(* CODESYS project AULA1.project

Project tree, tasks and I/O mapping:
  Device : CODESYS Control Win V3, 3S - Smart Software Solutions GmbH, order no. 305021, version 3.5.11.30
    application Application
      libraries: Standard, * (System)
      task MainTask (cyclic, interval t#20ms, priority 1) calls PLC_PRG
      task VISU_TASK (cyclic, interval 100 ms, priority 31) calls VisuElems.Visu_Prg
      program PLC_PRG [LD]
      visualisation Visualization
  text list GlobalTextList
*)

// Device/Application/PLC_PRG
PROGRAM PLC_PRG
VAR
	A : BOOL;
	B : BOOL;
	C : BOOL;
	SNOT: BOOL;
	SOR: BOOL;
	SAND2: BOOL;
	SAND1: BOOL;
	SA : BOOL;
END_VAR

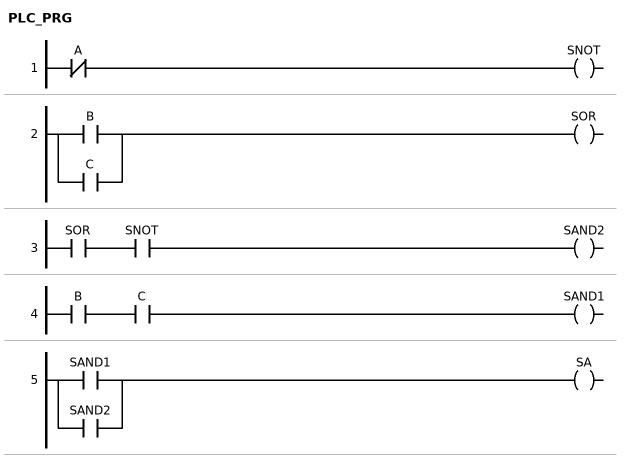
// NETWORK 1
SNOT := NOT A;

// NETWORK 2
SOR := B OR C;

// NETWORK 3
SAND2 := SOR AND SNOT;

// NETWORK 4
SAND1 := B AND C;

// NETWORK 5
SA := SAND1 OR SAND2;

END_PROGRAM

// Device/Application/Visualization
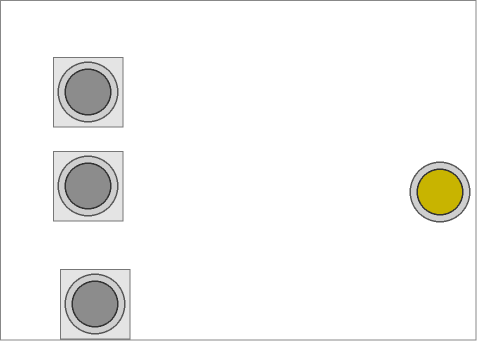
VISUALIZATION Visualization  // 477x341
    Lamp1 (405,157 70x70), variable: PLC_PRG.SA, style: Lamp-Lamp1-Yellow
    PushSwitchLed (53,57 70x70), variable: PLC_PRG.A, behaviour: TOGGLE, style: Switch-PushSwitchLed-Gray
    PushSwitchLed (53,151 70x70), variable: PLC_PRG.B, behaviour: TOGGLE, style: Switch-PushSwitchLed-Gray
    PushSwitchLed (60,269 70x70), variable: PLC_PRG.C, behaviour: TOGGLE, style: Switch-PushSwitchLed-Gray
END_VISUALIZATION
